// TIA Portal project "LAVADER0 DE COCHES" (V11)

(* hardware
DEVICE "S7300/ET200 station_1"  SIMATIC 300-Station
   slot 0: "Perfil soporte_0"  Rail  6ES7 390-1***0-0AA0
   slot 2: "PLC_1"  CPU 313C-2 DP  6ES7 313-6CF03-0AB0  V2.6
      slot 0: "Interfaz MPI_1"  MPI
      slot 1: "Interfaz DP_1"  DP
      slot 2: "DI16/DO16_1"  DI16/DO16
      slot 4: "Contaje_1"  Counter
DEVICE "S7300/ET200 station_2"  SIMATIC 300-Station
   slot 0: "Perfil soporte_0"  Rail  6ES7 390-1***0-0AA0
   slot 2: "JAVA"  CPU 313C-2 DP  6ES7 313-6CF03-0AB0  V2.6
      slot 0: "Interfaz MPI_1"  MPI
      slot 1: "Interfaz DP_1"  DP
      slot 2: "DI16/DO16_1"  DI16/DO16
      slot 4: "Contaje_1"  Counter
*)

// ===== PLC "PLC_1"  CPU 313C-2 DP =====

VAR_GLOBAL   // PLC tag table "Tabla de variables estándar"
   "M1 KM1 D ARRASTRE LENTA" AT %A0.0 : Bool;
   "M1 KM2 D ARRASTRE RAPIDA" AT %A0.1 : Bool;
   "M1 KM3 COMUN RAPIDA" AT %A0.2 : Bool;
   "M1 KM4 I RETROCESO LENTA" AT %A0.3 : Bool;
   "M1 KM5 I RETROCESO RAPIDA" AT %A0.4 : Bool;
   "M2 D VERTICAL" AT %A0.5 : Bool;
   "M2 I VERTICAL" AT %A0.6 : Bool;
   "M3 D HORIZONTAL" AT %A0.7 : Bool;
   "M3 I HORIZONTAL" AT %A1.0 : Bool;
   "M4 D LAVADO RUEDAS" AT %A1.1 : Bool;
   "M4 I LAVADO RUEDAS" AT %A1.2 : Bool;
   "VENTILADOR LINEA" AT %A1.3 : Bool;
   "VENTILADOE ESTRELLA" AT %A1.4 : Bool;
   "VENTILDOR TRIANGULO" AT %A1.5 : Bool;
   "BOMBA AGUA" AT %A1.6 : Bool;
   "BOMBA AIRE" AT %A1.7 : Bool;
   "BOMBA CHAMPU" AT %A2.0 : Bool;
   "tag_18" AT %E0.0 : Bool;
   "tag_19" AT %E0.1 : Bool;
   "tag_20" AT %E0.2 : Bool;
   "tag_21" AT %E0.3 : Bool;
   "Tag_22" AT %E0.4 : Bool;
   "Tag_23" AT %E0.5 : Bool;
   "Tag_24" AT %E0.6 : Bool;
   "Tag_25" AT %E0.7 : Bool;
   "Tag_26" AT %E1.0 : Bool;
   "Tag_27" AT %E1.1 : Bool;
   "Tag_28" AT %E1.2 : Bool;
   "Tag_29" AT %E1.3 : Bool;
   "Tag_30" AT %E1.4 : Bool;
   "Tag_31" AT %E1.5 : Bool;
   "Tag_32" AT %E1.6 : Bool;
   "Tag_33" AT %E1.7 : Bool;
   "tag_34" AT %E2.0 : Bool;
   "BOMBA CERA" AT %A2.1 : Bool;
   "PISTON VERTICAL" AT %A2.2 : Bool;
   "PISTON HORIZONTAL" AT %A2.3 : Bool;
   "PISTON L RUEDAS" AT %A2.4 : Bool;
   "Tag_39" AT %M0.0 : Bool;
   "Tag_1" AT %M0.3 : Bool;
   "Tag_2" AT %M0.4 : Bool;
   "Tag_3" AT %M0.5 : Bool;
   "Tag_4" AT %M0.6 : Bool;
   "Tag_5" AT %M0.7 : Bool;
   "Tag_6" AT %A11.5 : Bool;
   "Tag_7" AT %M8.0 : Bool;
   "Tag_8" AT %M10.0 : Bool;
   "Tag_9" AT %M10.1 : Bool;
   "Tag_10" AT %E2.2 : Bool;
   "V V EXPANDIDO" AT %A2.5 : Bool;
   "V V CONTRAIDO" AT %A2.6 : Bool;
   "V V SEMICONTRIDO" AT %A2.7 : Bool;
END_VAR

DATA_BLOCK "LAVADERO_DB"   // DB1
{ S7_Optimized_Access := 'FALSE' }
VERSION : 0.1
// stored: InstanceOfName LAVADERO
"LAVADERO"
BEGIN
   SWITCH[0] := 16#0;
   SW_SQTS[0] := 16#19;
   SW_SQTS[1] := 16#0;
   SW_SQTS[2] := 16#1;
   SW_SQTS[3] := 16#2;
   SW_SQTS[4] := 16#3;
   TVX[0] := 16#1;
   TTX[0] := 16#1;
   TSX[0] := 16#1;
   S00X[0] := 16#1;
   SOFFX[0] := 16#1;
   SONX[0] := 16#1;
   SAX[0] := 16#1;
   SERRX[0] := 16#1;
   SMX[0] := 16#1;
   S0X[0] := 16#1;
   S1X[0] := 16#1;
   SINI[0] := 16#2;
   SINI[1] := 16#1;
   LSTT[6] := 0;
   LSTT[5] := 16#1;
   ATAJ[1] := 16#1;
   ATAJ[2] := 16#2;
   ATAJ[3] := 16#3;
   ATAJ[4] := 16#4;
   ATAJ[5] := 16#5;
   ATAJ[6] := 16#6;
   ATAB[1] := 16#1B;
   ATAB[2] := 16#3;
   ATAB[3] := 16#1;
   ATAB[4] := 16#4;
   ATAB[5] := 16#5;
   ATAB[6] := 16#7;
   PSTT[1] := 16#1;
   PSTT[2] := 16#1;
   PSTT[3] := 16#1;
   PSTT[4] := 16#2;
   PSTT[5] := 16#3;
   PSTT[6] := 16#4;
   NSTT[0] := 16#1;
   NSTT[1] := 16#4;
   NSTT[2] := 16#2;
   NSTT[3] := 16#3;
   NSTT[4] := 16#1;
   NSTT[5] := 16#1;
   NSTT[6] := 16#5;
   ASSJ[1] := 16#1;
   ASSJ[2] := 16#2;
   ASSJ[3] := 16#3;
   ASSJ[4] := 16#4;
   ASSB[1] := 16#1;
   ASSB[2] := 16#2;
   ASSB[3] := 16#3;
   ASSB[4] := 16#4;
   PTTS[1] := 16#0;
   PTTS[2] := 16#2;
   PTTS[3] := 16#3;
   PTTS[4] := 16#1;
   NTTS[1] := 16#1;
   NTTS[2] := 16#4;
   NTTS[3] := 16#5;
   NTTS[4] := 16#6;
   LSTT[4] := 16#1;
   ATAJ[7] := 16#7;
   ATAB[7] := 16#6;
   PSTT[7] := 16#4;
   NSTT[7] := 16#1;
   SW_SQTS[5] := 16#4;
   ASSJ[5] := 16#5;
   ASSB[5] := 16#B;
   PTTS[5] := 16#6;
   NTTS[5] := 16#A;
   LSTT[7] := 16#1;
   SWITCH[1] := 16#0;
   SW_SQTS[6] := 16#5;
   SW_SQTS[7] := 16#6;
   LSTT[9] := 0;
   LSTT[10] := 0;
   ATAJ[8] := 16#8;
   ATAJ[9] := 16#9;
   ATAJ[10] := 16#A;
   ATAB[8] := 16#14;
   ATAB[9] := 16#D;
   ATAB[10] := 16#C;
   PSTT[8] := 16#8;
   PSTT[9] := 16#6;
   PSTT[10] := 16#5;
   NSTT[8] := 16#F;
   NSTT[9] := 16#7;
   NSTT[10] := 16#6;
   ASSJ[6] := 16#6;
   ASSJ[7] := 16#7;
   ASSB[6] := 16#6;
   ASSB[7] := 16#7;
   PTTS[6] := 16#A;
   PTTS[7] := 16#9;
   NTTS[6] := 16#9;
   NTTS[7] := 16#B;
   LSTT[11] := 0;
   ATAJ[11] := 16#B;
   ATAB[11] := 16#F;
   PSTT[11] := 16#7;
   NSTT[11] := 16#8;
   ATAJ[12] := 16#C;
   ATAB[12] := 16#A;
   PSTT[12] := 16#5;
   NSTT[12] := 16#1;
   LSTT[8] := 0;
   SW_SQTS[8] := 16#7;
   ASSJ[8] := 16#8;
   ASSB[8] := 16#8;
   PTTS[8] := 16#B;
   NTTS[8] := 16#8;
   LSTT[12] := 16#1;
   SWITCH[2] := 16#0;
   SW_SQTS[9] := 16#8;
   ATAJ[13] := 16#D;
   ATAB[13] := 16#9;
   PSTT[13] := 16#6;
   NSTT[13] := 16#1;
   ASSJ[9] := 16#9;
   ASSB[9] := 16#9;
   PTTS[9] := 16#E;
   NTTS[9] := 16#11;
   SWITCH[3] := 16#400106;
   SW_SQTS[10] := 16#9;
   LSTT[15] := 16#1;
   LSTT[16] := 16#1;
   LSTT[18] := 0;
   LSTT[19] := 16#13;
   ATAJ[14] := 16#E;
   ATAJ[15] := 16#F;
   ATAJ[16] := 16#10;
   ATAJ[17] := 16#11;
   ATAJ[18] := 16#12;
   ATAJ[19] := 16#13;
   ATAB[14] := 16#10;
   ATAB[15] := 16#B;
   ATAB[16] := 16#E;
   ATAB[17] := 16#15;
   ATAB[18] := 16#20;
   ATAB[19] := 16#17;
   PSTT[14] := 16#F;
   PSTT[15] := 16#7;
   PSTT[16] := 16#F;
   PSTT[17] := 16#9;
   PSTT[18] := 16#12;
   PSTT[19] := 16#C;
   NSTT[14] := 16#9;
   NSTT[15] := 16#1;
   NSTT[16] := 16#1;
   NSTT[17] := 16#A;
   NSTT[18] := 16#C;
   NSTT[19] := 16#13;
   ASSJ[10] := 16#A;
   ASSB[10] := 16#A;
   PTTS[10] := 16#11;
   NTTS[10] := 16#1F;
   SWITCH[4] := 16#80020C00;
   SW_SQTS[11] := 16#A;
   SW_SQTS[12] := 16#B;
   SW_SQTS[13] := 16#C;
   ATAJ[20] := 16#14;
   ATAJ[21] := 16#15;
   ATAB[20] := 16#8;
   ATAB[21] := 16#11;
   PSTT[20] := 16#8;
   PSTT[21] := 16#9;
   NSTT[20] := 16#1;
   NSTT[21] := 16#1;
   ASSJ[11] := 16#B;
   ASSJ[12] := 16#C;
   ASSJ[13] := 16#D;
   ASSB[11] := 16#16;
   ASSB[12] := 16#C;
   ASSB[13] := 16#D;
   PTTS[11] := 16#6;
   PTTS[12] := 16#12;
   PTTS[13] := 16#18;
   NTTS[11] := 16#18;
   NTTS[12] := 16#13;
   NTTS[13] := 16#19;
   SWITCH[5] := 16#518000A;
   SWITCH[6] := 16#30001460;
   SW_SQTS[14] := 16#D;
   LSTT[23] := 16#1;
   LSTT[24] := 0;
   LSTT[25] := 16#B;
   ATAJ[22] := 16#16;
   ATAJ[23] := 16#17;
   ATAJ[24] := 16#18;
   ATAJ[25] := 16#19;
   ATAB[22] := 16#1F;
   ATAB[23] := 16#13;
   ATAB[24] := 16#1A;
   ATAB[25] := 16#19;
   PSTT[22] := 16#A;
   PSTT[23] := 16#C;
   PSTT[24] := 16#B;
   PSTT[25] := 16#D;
   NSTT[22] := 16#1;
   NSTT[23] := 16#1;
   NSTT[24] := 16#D;
   NSTT[25] := 16#B;
   ASSJ[14] := 16#E;
   ASSB[14] := 16#10;
   PTTS[14] := 16#22;
   NTTS[14] := 16#1C;
   SWITCH[7] := 16#28C0C0;
   SW_SQTS[15] := 16#E;
   ATAJ[26] := 16#1A;
   ATAB[26] := 16#18;
   PSTT[26] := 16#B;
   NSTT[26] := 16#1;
   ASSJ[15] := 16#F;
   ASSB[15] := 16#F;
   PTTS[15] := 16#8;
   NTTS[15] := 16#E;
   LSTT[27] := 0;
   ATAJ[27] := 16#1B;
   ATAB[27] := 16#2;
   PSTT[27] := 16#1;
   NSTT[27] := 16#13;
   SW_SQTS[16] := 16#F;
   ATAJ[28] := 16#1C;
   ATAB[28] := 16#2C;
   PSTT[28] := 16#E;
   NSTT[28] := 16#14;
   ASSJ[16] := 16#10;
   ASSB[16] := 16#18;
   PTTS[16] := 16#22;
   NTTS[16] := 16#1D;
   LSTT[29] := 0;
   ATAJ[29] := 16#1D;
   ATAB[29] := 16#21;
   PSTT[29] := 16#10;
   NSTT[29] := 16#11;
   LSTT[26] := 16#1;
   LSTT[30] := 16#10;
   ATAJ[30] := 16#1E;
   ATAB[30] := 16#1E;
   PSTT[30] := 16#11;
   NSTT[30] := 16#10;
   SWITCH[8] := 16#2F8901A0;
   SWITCH[9] := 16#3BF24;
   SW_SQTS[17] := 16#10;
   LSTT[32] := 16#1;
   ATAJ[31] := 16#1F;
   ATAJ[32] := 16#20;
   ATAB[31] := 16#16;
   ATAB[32] := 16#12;
   PSTT[31] := 16#A;
   PSTT[32] := 16#12;
   NSTT[31] := 16#12;
   NSTT[32] := 16#1;
   ASSJ[17] := 16#11;
   ASSB[17] := 16#11;
   PTTS[17] := 16#1D;
   NTTS[17] := 16#1E;
   SW_SQTS[18] := 16#11;
   LSTT[17] := 0;
   LSTT[20] := 16#1;
   LSTT[28] := 0;
   LSTT[31] := 0;
   LSTT[33] := 16#1;
   ATAJ[33] := 16#21;
   ATAB[33] := 16#1D;
   PSTT[33] := 16#10;
   NSTT[33] := 16#1;
   ASSJ[18] := 16#12;
   ASSB[18] := 16#12;
   PTTS[18] := 16#1F;
   NTTS[18] := 16#12;
   SWITCH[10] := 16#6003030;
   LSTT[34] := 0;
   ATAJ[34] := 16#22;
   ATAB[34] := 16#23;
   PSTT[34] := 16#13;
   NSTT[34] := 16#E;
   SWITCH[11] := 16#51800;
   SW_SQTS[19] := 16#12;
   SW_SQTS[20] := 16#13;
   LSTT[36] := 16#1;
   LSTT[37] := 0;
   ATAJ[35] := 16#23;
   ATAJ[36] := 16#24;
   ATAJ[37] := 16#25;
   ATAB[35] := 16#22;
   ATAB[36] := 16#24;
   ATAB[37] := 16#2D;
   PSTT[35] := 16#13;
   PSTT[36] := 16#15;
   PSTT[37] := 16#14;
   NSTT[35] := 16#1;
   NSTT[36] := 16#1;
   NSTT[37] := 16#15;
   ASSJ[19] := 16#13;
   ASSJ[20] := 16#14;
   ASSB[19] := 16#13;
   ASSB[20] := 16#14;
   PTTS[19] := 16#1B;
   PTTS[20] := 16#1C;
   NTTS[19] := 16#22;
   NTTS[20] := 16#25;
   SW_SQTS[21] := 16#14;
   ATAJ[38] := 16#26;
   ATAB[38] := 16#28;
   PSTT[38] := 16#16;
   NSTT[38] := 16#17;
   ASSJ[21] := 16#15;
   ASSB[21] := 16#15;
   PTTS[21] := 16#25;
   NTTS[21] := 16#24;
   SWITCH[12] := 16#10CC0020;
   SWITCH[13] := 16#980128C0;
   LSTT[38] := 0;
   LSTT[39] := 16#16;
   ATAJ[39] := 16#27;
   ATAB[39] := 16#27;
   PSTT[39] := 16#17;
   NSTT[39] := 16#16;
   SW_SQTS[22] := 16#15;
   SW_SQTS[23] := 16#16;
   LSTT[40] := 16#1;
   ATAJ[40] := 16#28;
   ATAB[40] := 16#26;
   PSTT[40] := 16#16;
   NSTT[40] := 16#1;
   ASSJ[22] := 16#16;
   ASSJ[23] := 16#17;
   ASSB[22] := 16#5;
   ASSB[23] := 16#17;
   PTTS[22] := 16#6;
   PTTS[23] := 16#26;
   NTTS[22] := 16#26;
   NTTS[23] := 16#27;
   LSTT[35] := 16#1;
   LSTT[22] := 16#1;
   LSTT[21] := 16#1;
   LSTT[13] := 16#1;
   SWITCH[14] := 16#0;
   SWITCH[15] := 16#C0C00;
   SWITCH[16] := 16#1818FE4B;
   SW_SQTS[24] := 16#17;
   SW_SQTS[25] := 16#18;
   LSTT[42] := 16#18;
   LSTT[43] := 16#1;
   ATAJ[41] := 16#29;
   ATAJ[42] := 16#2A;
   ATAJ[43] := 16#2B;
   ATAB[41] := 16#2B;
   ATAB[42] := 16#2A;
   ATAB[43] := 16#29;
   PSTT[41] := 16#18;
   PSTT[42] := 16#19;
   PSTT[43] := 16#18;
   NSTT[41] := 16#19;
   NSTT[42] := 16#18;
   NSTT[43] := 16#1;
   ASSJ[24] := 16#18;
   ASSJ[25] := 16#19;
   ASSB[24] := 16#E;
   ASSB[25] := 16#19;
   PTTS[24] := 16#22;
   PTTS[25] := 16#29;
   NTTS[24] := 16#29;
   NTTS[25] := 16#2A;
   SWITCH[17] := 16#FC9700;
   SWITCH[18] := 16#D00C00;
   SWITCH[19] := 16#A0190000;
   LSTT[44] := 16#1;
   LSTT[45] := 16#1;
   ATAJ[44] := 16#2C;
   ATAJ[45] := 16#2D;
   ATAB[44] := 16#1C;
   ATAB[45] := 16#25;
   PSTT[44] := 16#E;
   PSTT[45] := 16#14;
   NSTT[44] := 16#1;
   NSTT[45] := 16#1;
END_DATA_BLOCK

FUNCTION_BLOCK "LAVADERO"   // FB1, GRAPH
{ S7_Optimized_Access := 'FALSE' }
VERSION : 0.1
   VAR_INPUT
      OFF_SQ : Bool := false;   // Desconectar cadena
      INIT_SQ : Bool := false;   // Poner cadena en estado inicial
      ACK_EF : Bool := false;   // Acusar todos los errores y fallos
      S_PREV : Bool := false;   // Mostrar la etapa anterior en el parámetro S_NO
      S_NEXT : Bool := false;   // Mostrar la etapa siguiente en el parámetro S_NO
      SW_AUTO : Bool := false;   // Modo automático
      SW_TAP : Bool := false;   // Semiautomático/continuar con transición
      SW_TOP : Bool := false;   // Semiautomático/transición ignorada
      SW_MAN : Bool := false;   // Modo manual
      S_SEL : Int := 0;   // Seleccionar la etapa que debe mostrarse en S_NO
      S_ON : Bool := false;   // Activar la etapa del parámetro S_NO
      S_OFF : Bool := false;   // Desactivar el incremento presente en el parámetro S_NO
      T_PUSH : Bool := false;   // Habilitar transición en modo semiautomático
      MICRO : Bool;
      SETA : Bool;
      EMERGENCIA : Bool;
      LLAVE : Bool;
      "A.CEPILLOS" : Bool;
      "S CEPILLOS" : Bool;
      "ABANCE CARRO" : Bool;
      "RETROCESO CARRO" : Bool;
      "FC LEVA" : Bool;
      "FC ABANCE" : Bool;
      "FC RETOCESO" : Bool;
      "FC VARILLA 1" : Bool;
      "SENSOR METALICO" : Bool;
      CLINOMETRO : Bool;
      CELULA : Bool;
   END_VAR
   VAR_OUTPUT
      S_NO : Int := 0;   // Número de etapa
      S_MORE : Bool := false;   // Existen más etapas que pueden mostrarse en S_NO.
      S_ACTIVE : Bool := false;   // El incremento presente en el parámetro S_NO está activo
      ERR_FLT : Bool := false;   // Error de grupo interlock o supervisión
      AUTO_ON : Bool := false;   // Modo automático activado
      TAP_ON : Bool := false;   // Modo semiautomático/etapa con transición activada
      TOP_ON : Bool := false;   // Modo semiautomático/Ignorar transición activado
      MAN_ON : Bool := false;   // Modo manual activado
      "M1 KM1 D ARRASTRE LENTA" : Bool;
      "M1 KM2 D ARRASTRE RAPIDA" : Bool;
      "M1 KM3 COMUN RAPIDA" : Bool;
      "M1 KM4 I RETROCESO LENTA" : Bool;
      "M1 KM5 I RETROCESO RAPIDA" : Bool;
      "M2 D VERTICAL" : Bool;
      "M2 I VERTICAL" : Bool;
      "M3 D HORIZONTAL" : Bool;
      "M3 I HORIZONTAL" : Bool;
      "M4 D LAVADO RUEDAS" : Bool;
      "M4 I LAVADO RUEDAS" : Bool;
      "VENTILADOR LINEA" : Bool;
      "VENTILADOR ESTRELLA" : Bool;
      "VENTILADOR TRIANULO" : Bool;
      "BOMBA AGUA" : Bool;
      "BOMBA AIRE" : Bool;
      "BOMBA CHAMPU" : Bool;
      "BOMBA CERA" : Bool;
      "PISTON VERTICAL" : Bool;
      "PISTON HORIZONAL" : Bool;
      "PISTON L RUEDAS" : Bool;
      "V V  EXPANDIDO" : Bool;
      "V V  CONTRAIDO" : Bool;
      "V V SEMICONTRAIDO" : Bool;
   END_VAR
   VAR
      SWITCH : Array [0..19]of DWord;
      SW_SQTS : Array [0..25]of Byte;
      SW_ADDR : Word := 16#E;
      G7T_0 : GraphTransition;
      G7S_0 : GraphStep;
      PRE_CRIT : Array [0..0]of DWord;
      POST_CRIT : Array [0..0]of DWord;
      TVX : Array [0..46]of Byte;
      TTX : Array [0..46]of Byte;
      TSX : Array [0..8]of Byte;
      S00X : Array [0..8]of Byte;
      SOFFX : Array [0..8]of Byte;
      SONX : Array [0..8]of Byte;
      SAX : Array [0..8]of Byte;
      SERRX : Array [0..26]of Byte;
      SMX : Array [0..26]of Byte;
      S0X : Array [0..26]of Byte;
      S1X : Array [0..26]of Byte;
      S_DISPLAY : Int;   // Indicación interna del parámetro de salida S_NO
      S_SEL_OLD : Int;   // Valor anterior en S_SEL
      S_DISPIDX : Byte;   // Índice de la etapa presente en S_NO
      T_DISPIDX : Byte;   // Índice de la transición presente en T_NO
      MOPEDGE : Struct
         AUTO : Bool := false;
         MAN : Bool := false;
         TAP : Bool := false;
         TOP : Bool := false;
         ACK_S : Bool := false;
         REG_S : Bool := false;
         T_PREV : Bool := false;
         T_NEXT : Bool := false;
         LOCK : Bool := false;
         SUP : Bool := false;
         ACKREQ : Bool := false;
         SSKIP : Bool := false;
         OFF : Bool := false;
         INIT : Bool := false;
         HALT : Bool := false;
         TMS_HALT : Bool := false;
         OPS_ZERO : Bool := false;
         SACT_DISP : Bool := false;
         SEF_DISP : Bool := false;
         SALL_DISP : Bool := false;
         S_PREV : Bool := false;
         S_NEXT : Bool := false;
         S_SELOK : Bool := false;
         S_ON : Bool := false;
         S_OFF : Bool := false;
         T_PUSH : Bool := false;
         REG : Bool := false;
         ACK : Bool := false;
         IL_PERM : Bool := false;
         T_PERM : Bool := false;
         ILP_MAN : Bool := false;
      END_STRUCT;
      MOP : Struct   // Modo de operación
         AUTO : Bool := true;   // Estado: modo automático
         MAN : Bool := false;   // Estado: modo manual
         TAP : Bool := false;   // Estado: semiautomático/continuar con transición
         TOP : Bool := false;   // Estado: semiautomático/transición ignorada
         ACK_S : Bool := false;   // Solicitud: acusar la etapa presente en el parámetro S_NO
         REG_S : Bool := false;   // Solicitud: registrar la etapa presente en el parámetro S_NO
         T_PREV : Bool := false;   // Solicitud: mostrar la transición anterior válida en el parámetro T_NO
         T_NEXT : Bool := false;   // Solicitud: mostrar la siguiente transición válida en el parámetro T_NO
         LOCK : Bool := true;   // Estado: ejecución de interlock activada
         SUP : Bool := true;   // Estado: ejecución de supervisión activada
         ACKREQ : Bool := true;   // Estado: acuse requerido
         SSKIP : Bool := false;   // Estado: "Saltar etapas" activado
         OFF : Bool := false;   // Solicitud: desactivar todas las etapas
         INIT : Bool := true;   // Solicitud: poner cadena en estado inicial
         HALT : Bool := false;   // Estado: la cadena no continúa
         TMS_HALT : Bool := false;   // Estado: todos los temporizadores internos detenidos
         OPS_ZERO : Bool := false;   // Estado: todos los operandos ejecutados con N, L, D puestos a 0
         SACT_DISP : Bool := true;   // Estado: mostrar sólo etapas activas
         SEF_DISP : Bool := false;   // Estado: mostrar sólo etapas erróneas y defectuosas
         SALL_DISP : Bool := false;   // Estado: mostrar todas las etapas
         S_PREV : Bool := false;   // Solicitud: mostrar la etapa anterior en el parámetro S_NO
         S_NEXT : Bool := false;   // Solicitud: Indicar etapa siguiente en el parámetro S_NO
         S_SELOK : Bool := false;   // Solicitud: mostrar en el parámetro S_NO el número de la etapa presente en el parámetro S_SEL
         S_ON : Bool := false;   // Solicitud: activar la etapa presente en el parámetro S_NO
         S_OFF : Bool := false;   // Solicitud: desactivar la etapa presente en el parámetro S_NO
         T_PUSH : Bool := false;   // Solicitud: habilitar transición
         REG : Bool := false;   // Solicitud: registrar todos los errores de interlock y supervisión
         ACK : Bool := false;   // Solicitud: acusar todos los errores de interlock y supervisión
         IL_PERM : Bool := false;   // Estado: ejecución permanente de todos los interlocks
         T_PERM : Bool := false;   // Estado: ejecución permanente de todas las transiciones
         ILP_MAN : Bool := false;   // Estado: ejecución permanente de todos los interlocks en modo manual
      END_STRUCT;
      TICKS : Struct   // Ciclos de tiempo
         DELTA : Time := T#0ms;   // Diferencia de tiempo entre dos ciclos
         OLD : Time := T#0ms;   // Estado de contador cíclico 10 ms en el último ciclo
         NEW : Time := T#0ms;   // Estado de contador cíclico 10 ms en este ciclo
      END_STRUCT;
      SQ_FLAGS : Struct   // Marcas de cadena
         ERR_FLT : Bool := false;   // Error de grupo interlock y supervisión
         ERROR : Bool := false;   // Error de grupo Interlock
         FAULT : Bool := false;   // Error de grupo Supervisión
         RT_FAIL : Bool := false;   // Error en tiempo de ejecución
         NO_SNO : Bool := false;   // No se ha encontrado el número de etapa solicitado
         NF_OFL : Bool := false;   // Desbordamiento: demasiadas solicitudes ON u OFF
         SA_OFL : Bool := false;   // Desbordamiento: demasiadas etapas activas
         TV_OFL : Bool := false;   // Desbordamiento: demasiadas transiciones válidas
         MSG_OFL : Bool := false;   // Desbordamiento: los recursos del sistema no son suficientes para ALARM_S
         NO_SWI : Bool := false;   // No conmutar en este ciclo
         CYC_OP : Bool := false;   // Ejecución cíclica de la cadena tras la inicialización
         AS_MSG : Bool := true;   // Avisos en tiempo de ejecución activados o desactivados por instrucción
         AS_SEND : Bool := false;   // Enviar avisos de WR_USMSG o sólo registrarlos en el búfer de diagnóstico
         SQ_BUSY : Bool := false;   // Marca de flanco interna para ejecución de proceso
         SA_BUSY : Bool := false;   // Marca de flanco interna para ejecución de proceso
         AS_SIG : Bool := false;   // Marca de flanco para avisos de Alarm_S y Alarm_SQ
      END_STRUCT;
      S_PTR : DWord := 16#1AD0;
      S_PTR2 : DWord := 16#0;
      S_PTR3 : DWord := 16#3C40;
      S_PTR4 : DWord := 16#3B60;
      T_PTR : DWord := 16#3A80;
      C_AR2 : DWord := 16#0;
      M_FBDB : DWord := 16#10000;
      M_SNO : Word := 16#0;
      M_EVID : Word := 16#0;
      M_EVIL : C_Alarm_s;
      M_EVSV : C_Alarm_s;
      M_EV : DWord := 16#38B0;
      CRIT : Array [0..31]of Bool;
      S_START : Byte := 16#0;
      S_IDX : Byte := 16#0;
      S_INT : Int := 72;
      S_TMP : Byte := 16#0;
      T_START : Byte := 16#0;
      T_IDX : Byte := 16#0;
      T_TMP : Byte := 16#0;
      T_TMP2 : Byte := 16#00;
      TV_POT : Byte := 16#08;
      RETURN1 : Byte := 16#0;
      RETURN2 : Byte := 16#0;
      SINI : Array [0..8]of Byte;
      LSTT : Array [0..45]of Byte;
      ATAJ : Array [0..45]of Byte;
      ATAB : Array [0..45]of Byte;
      PSTT : Array [0..45]of Byte;
      NSTT : Array [0..45]of Byte;
      ASSJ : Array [0..25]of Byte;
      ASSB : Array [0..25]of Byte;
      PTTS : Array [0..25]of Byte;
      NTTS : Array [0..25]of Byte;
      PRE_CNT : Word := 16#1;
      POST_CNT : Word := 16#1;
      ADR_COND : Word := 16#0;
      MAX_TVAL : Byte := 16#2D;
      MAX_SACT : Byte := 16#7;
      MAX_CRIT : Byte := 16#4;
      T_CNT : Byte := 16#2D;
      SUP_CNT : Byte := 16#0;
      LOCK_CNT : Byte := 16#6;
      S_CNT : Byte := 16#19;
      SQ_CNT : Byte := 16#1;
      PRS_INPAR : DWord := 16#E000FEC8;
      PRS_OUTPAR : DWord := 16#E000800F;
      GC_FLAGS : Struct
         T_MACH : Byte := 16#EB;
         COND_ED : Byte := 16#E3;
         W_LEVEL : Byte := 16#D5;
         FB_IF : Byte := 16#FA;
         AS_MSG : Word := 16#202;
         SSB : Word := 16#108;
         DILG : Word := 16#97C;
         ADDR_T0 : Word := 16#7A;
         CRIT_AVAIL : Bool := false;
         SSKIP_AVAIL : Bool := true;
         SSKIP_ON : Bool := false;
         ACK_REQ : Bool := true;
         SYNC_AVAIL : Bool := true;
         ILP_MAN : Bool := false;
         SWM_LOCKED : Bool := false;
         SAVE_SW : Bool := true;
      END_STRUCT;
      G7_FBMARK : Byte := 16#3C;
      G7_RELEASE : Byte := 16#3C;
      G7_ID2 : Byte := 16#37;
      G7_ID1 : Byte := 16#47;
   END_VAR
   // SWITCH[0] := 16#0;
   // SW_SQTS[0] := 16#19;
   // SW_SQTS[1] := 16#0;
   // SW_SQTS[2] := 16#1;
   // SW_SQTS[3] := 16#2;
   // SW_SQTS[4] := 16#3;
   // TVX[0] := 16#1;
   // TTX[0] := 16#1;
   // TSX[0] := 16#1;
   // S00X[0] := 16#1;
   // SOFFX[0] := 16#1;
   // SONX[0] := 16#1;
   // SAX[0] := 16#1;
   // SERRX[0] := 16#1;
   // SMX[0] := 16#1;
   // S0X[0] := 16#1;
   // S1X[0] := 16#1;
   // SINI[0] := 16#2;
   // SINI[1] := 16#1;
   // LSTT[6] := 0;
   // LSTT[5] := 16#1;
   // ATAJ[1] := 16#1;
   // ATAJ[2] := 16#2;
   // ATAJ[3] := 16#3;
   // ATAJ[4] := 16#4;
   // ATAJ[5] := 16#5;
   // ATAJ[6] := 16#6;
   // ATAB[1] := 16#1B;
   // ATAB[2] := 16#3;
   // ATAB[3] := 16#1;
   // ATAB[4] := 16#4;
   // ATAB[5] := 16#5;
   // ATAB[6] := 16#7;
   // PSTT[1] := 16#1;
   // PSTT[2] := 16#1;
   // PSTT[3] := 16#1;
   // PSTT[4] := 16#2;
   // PSTT[5] := 16#3;
   // PSTT[6] := 16#4;
   // NSTT[0] := 16#1;
   // NSTT[1] := 16#4;
   // NSTT[2] := 16#2;
   // NSTT[3] := 16#3;
   // NSTT[4] := 16#1;
   // NSTT[5] := 16#1;
   // NSTT[6] := 16#5;
   // ASSJ[1] := 16#1;
   // ASSJ[2] := 16#2;
   // ASSJ[3] := 16#3;
   // ASSJ[4] := 16#4;
   // ASSB[1] := 16#1;
   // ASSB[2] := 16#2;
   // ASSB[3] := 16#3;
   // ASSB[4] := 16#4;
   // PTTS[1] := 16#0;
   // PTTS[2] := 16#2;
   // PTTS[3] := 16#3;
   // PTTS[4] := 16#1;
   // NTTS[1] := 16#1;
   // NTTS[2] := 16#4;
   // NTTS[3] := 16#5;
   // NTTS[4] := 16#6;
   // LSTT[4] := 16#1;
   // ATAJ[7] := 16#7;
   // ATAB[7] := 16#6;
   // PSTT[7] := 16#4;
   // NSTT[7] := 16#1;
   // SW_SQTS[5] := 16#4;
   // ASSJ[5] := 16#5;
   // ASSB[5] := 16#B;
   // PTTS[5] := 16#6;
   // NTTS[5] := 16#A;
   // LSTT[7] := 16#1;
   // SWITCH[1] := 16#0;
   // SW_SQTS[6] := 16#5;
   // SW_SQTS[7] := 16#6;
   // LSTT[9] := 0;
   // LSTT[10] := 0;
   // ATAJ[8] := 16#8;
   // ATAJ[9] := 16#9;
   // ATAJ[10] := 16#A;
   // ATAB[8] := 16#14;
   // ATAB[9] := 16#D;
   // ATAB[10] := 16#C;
   // PSTT[8] := 16#8;
   // PSTT[9] := 16#6;
   // PSTT[10] := 16#5;
   // NSTT[8] := 16#F;
   // NSTT[9] := 16#7;
   // NSTT[10] := 16#6;
   // ASSJ[6] := 16#6;
   // ASSJ[7] := 16#7;
   // ASSB[6] := 16#6;
   // ASSB[7] := 16#7;
   // PTTS[6] := 16#A;
   // PTTS[7] := 16#9;
   // NTTS[6] := 16#9;
   // NTTS[7] := 16#B;
   // LSTT[11] := 0;
   // ATAJ[11] := 16#B;
   // ATAB[11] := 16#F;
   // PSTT[11] := 16#7;
   // NSTT[11] := 16#8;
   // ATAJ[12] := 16#C;
   // ATAB[12] := 16#A;
   // PSTT[12] := 16#5;
   // NSTT[12] := 16#1;
   // LSTT[8] := 0;
   // SW_SQTS[8] := 16#7;
   // ASSJ[8] := 16#8;
   // ASSB[8] := 16#8;
   // PTTS[8] := 16#B;
   // NTTS[8] := 16#8;
   // LSTT[12] := 16#1;
   // SWITCH[2] := 16#0;
   // SW_SQTS[9] := 16#8;
   // ATAJ[13] := 16#D;
   // ATAB[13] := 16#9;
   // PSTT[13] := 16#6;
   // NSTT[13] := 16#1;
   // ASSJ[9] := 16#9;
   // ASSB[9] := 16#9;
   // PTTS[9] := 16#E;
   // NTTS[9] := 16#11;
   // SWITCH[3] := 16#400106;
   // SW_SQTS[10] := 16#9;
   // LSTT[15] := 16#1;
   // LSTT[16] := 16#1;
   // LSTT[18] := 0;
   // LSTT[19] := 16#13;
   // ATAJ[14] := 16#E;
   // ATAJ[15] := 16#F;
   // ATAJ[16] := 16#10;
   // ATAJ[17] := 16#11;
   // ATAJ[18] := 16#12;
   // ATAJ[19] := 16#13;
   // ATAB[14] := 16#10;
   // ATAB[15] := 16#B;
   // ATAB[16] := 16#E;
   // ATAB[17] := 16#15;
   // ATAB[18] := 16#20;
   // ATAB[19] := 16#17;
   // PSTT[14] := 16#F;
   // PSTT[15] := 16#7;
   // PSTT[16] := 16#F;
   // PSTT[17] := 16#9;
   // PSTT[18] := 16#12;
   // PSTT[19] := 16#C;
   // NSTT[14] := 16#9;
   // NSTT[15] := 16#1;
   // NSTT[16] := 16#1;
   // NSTT[17] := 16#A;
   // NSTT[18] := 16#C;
   // NSTT[19] := 16#13;
   // ASSJ[10] := 16#A;
   // ASSB[10] := 16#A;
   // PTTS[10] := 16#11;
   // NTTS[10] := 16#1F;
   // SWITCH[4] := 16#80020C00;
   // SW_SQTS[11] := 16#A;
   // SW_SQTS[12] := 16#B;
   // SW_SQTS[13] := 16#C;
   // ATAJ[20] := 16#14;
   // ATAJ[21] := 16#15;
   // ATAB[20] := 16#8;
   // ATAB[21] := 16#11;
   // PSTT[20] := 16#8;
   // PSTT[21] := 16#9;
   // NSTT[20] := 16#1;
   // NSTT[21] := 16#1;
   // ASSJ[11] := 16#B;
   // ASSJ[12] := 16#C;
   // ASSJ[13] := 16#D;
   // ASSB[11] := 16#16;
   // ASSB[12] := 16#C;
   // ASSB[13] := 16#D;
   // PTTS[11] := 16#6;
   // PTTS[12] := 16#12;
   // PTTS[13] := 16#18;
   // NTTS[11] := 16#18;
   // NTTS[12] := 16#13;
   // NTTS[13] := 16#19;
   // SWITCH[5] := 16#518000A;
   // SWITCH[6] := 16#30001460;
   // SW_SQTS[14] := 16#D;
   // LSTT[23] := 16#1;
   // LSTT[24] := 0;
   // LSTT[25] := 16#B;
   // ATAJ[22] := 16#16;
   // ATAJ[23] := 16#17;
   // ATAJ[24] := 16#18;
   // ATAJ[25] := 16#19;
   // ATAB[22] := 16#1F;
   // ATAB[23] := 16#13;
   // ATAB[24] := 16#1A;
   // ATAB[25] := 16#19;
   // PSTT[22] := 16#A;
   // PSTT[23] := 16#C;
   // PSTT[24] := 16#B;
   // PSTT[25] := 16#D;
   // NSTT[22] := 16#1;
   // NSTT[23] := 16#1;
   // NSTT[24] := 16#D;
   // NSTT[25] := 16#B;
   // ASSJ[14] := 16#E;
   // ASSB[14] := 16#10;
   // PTTS[14] := 16#22;
   // NTTS[14] := 16#1C;
   // SWITCH[7] := 16#28C0C0;
   // SW_SQTS[15] := 16#E;
   // ATAJ[26] := 16#1A;
   // ATAB[26] := 16#18;
   // PSTT[26] := 16#B;
   // NSTT[26] := 16#1;
   // ASSJ[15] := 16#F;
   // ASSB[15] := 16#F;
   // PTTS[15] := 16#8;
   // NTTS[15] := 16#E;
   // LSTT[27] := 0;
   // ATAJ[27] := 16#1B;
   // ATAB[27] := 16#2;
   // PSTT[27] := 16#1;
   // NSTT[27] := 16#13;
   // SW_SQTS[16] := 16#F;
   // ATAJ[28] := 16#1C;
   // ATAB[28] := 16#2C;
   // PSTT[28] := 16#E;
   // NSTT[28] := 16#14;
   // ASSJ[16] := 16#10;
   // ASSB[16] := 16#18;
   // PTTS[16] := 16#22;
   // NTTS[16] := 16#1D;
   // LSTT[29] := 0;
   // ATAJ[29] := 16#1D;
   // ATAB[29] := 16#21;
   // PSTT[29] := 16#10;
   // NSTT[29] := 16#11;
   // LSTT[26] := 16#1;
   // LSTT[30] := 16#10;
   // ATAJ[30] := 16#1E;
   // ATAB[30] := 16#1E;
   // PSTT[30] := 16#11;
   // NSTT[30] := 16#10;
   // SWITCH[8] := 16#2F8901A0;
   // SWITCH[9] := 16#3BF24;
   // SW_SQTS[17] := 16#10;
   // LSTT[32] := 16#1;
   // ATAJ[31] := 16#1F;
   // ATAJ[32] := 16#20;
   // ATAB[31] := 16#16;
   // ATAB[32] := 16#12;
   // PSTT[31] := 16#A;
   // PSTT[32] := 16#12;
   // NSTT[31] := 16#12;
   // NSTT[32] := 16#1;
   // ASSJ[17] := 16#11;
   // ASSB[17] := 16#11;
   // PTTS[17] := 16#1D;
   // NTTS[17] := 16#1E;
   // SW_SQTS[18] := 16#11;
   // LSTT[17] := 0;
   // LSTT[20] := 16#1;
   // LSTT[28] := 0;
   // LSTT[31] := 0;
   // LSTT[33] := 16#1;
   // ATAJ[33] := 16#21;
   // ATAB[33] := 16#1D;
   // PSTT[33] := 16#10;
   // NSTT[33] := 16#1;
   // ASSJ[18] := 16#12;
   // ASSB[18] := 16#12;
   // PTTS[18] := 16#1F;
   // NTTS[18] := 16#12;
   // SWITCH[10] := 16#6003030;
   // LSTT[34] := 0;
   // ATAJ[34] := 16#22;
   // ATAB[34] := 16#23;
   // PSTT[34] := 16#13;
   // NSTT[34] := 16#E;
   // SWITCH[11] := 16#51800;
   // SW_SQTS[19] := 16#12;
   // SW_SQTS[20] := 16#13;
   // LSTT[36] := 16#1;
   // LSTT[37] := 0;
   // ATAJ[35] := 16#23;
   // ATAJ[36] := 16#24;
   // ATAJ[37] := 16#25;
   // ATAB[35] := 16#22;
   // ATAB[36] := 16#24;
   // ATAB[37] := 16#2D;
   // PSTT[35] := 16#13;
   // PSTT[36] := 16#15;
   // PSTT[37] := 16#14;
   // NSTT[35] := 16#1;
   // NSTT[36] := 16#1;
   // NSTT[37] := 16#15;
   // ASSJ[19] := 16#13;
   // ASSJ[20] := 16#14;
   // ASSB[19] := 16#13;
   // ASSB[20] := 16#14;
   // PTTS[19] := 16#1B;
   // PTTS[20] := 16#1C;
   // NTTS[19] := 16#22;
   // NTTS[20] := 16#25;
   // SW_SQTS[21] := 16#14;
   // ATAJ[38] := 16#26;
   // ATAB[38] := 16#28;
   // PSTT[38] := 16#16;
   // NSTT[38] := 16#17;
   // ASSJ[21] := 16#15;
   // ASSB[21] := 16#15;
   // PTTS[21] := 16#25;
   // NTTS[21] := 16#24;
   // SWITCH[12] := 16#10CC0020;
   // SWITCH[13] := 16#980128C0;
   // LSTT[38] := 0;
   // LSTT[39] := 16#16;
   // ATAJ[39] := 16#27;
   // ATAB[39] := 16#27;
   // PSTT[39] := 16#17;
   // NSTT[39] := 16#16;
   // SW_SQTS[22] := 16#15;
   // SW_SQTS[23] := 16#16;
   // LSTT[40] := 16#1;
   // ATAJ[40] := 16#28;
   // ATAB[40] := 16#26;
   // PSTT[40] := 16#16;
   // NSTT[40] := 16#1;
   // ASSJ[22] := 16#16;
   // ASSJ[23] := 16#17;
   // ASSB[22] := 16#5;
   // ASSB[23] := 16#17;
   // PTTS[22] := 16#6;
   // PTTS[23] := 16#26;
   // NTTS[22] := 16#26;
   // NTTS[23] := 16#27;
   // LSTT[35] := 16#1;
   // LSTT[22] := 16#1;
   // LSTT[21] := 16#1;
   // LSTT[13] := 16#1;
   // SWITCH[14] := 16#0;
   // SWITCH[15] := 16#C0C00;
   // SWITCH[16] := 16#1818FE4B;
   // SW_SQTS[24] := 16#17;
   // SW_SQTS[25] := 16#18;
   // LSTT[42] := 16#18;
   // LSTT[43] := 16#1;
   // ATAJ[41] := 16#29;
   // ATAJ[42] := 16#2A;
   // ATAJ[43] := 16#2B;
   // ATAB[41] := 16#2B;
   // ATAB[42] := 16#2A;
   // ATAB[43] := 16#29;
   // PSTT[41] := 16#18;
   // PSTT[42] := 16#19;
   // PSTT[43] := 16#18;
   // NSTT[41] := 16#19;
   // NSTT[42] := 16#18;
   // NSTT[43] := 16#1;
   // ASSJ[24] := 16#18;
   // ASSJ[25] := 16#19;
   // ASSB[24] := 16#E;
   // ASSB[25] := 16#19;
   // PTTS[24] := 16#22;
   // PTTS[25] := 16#29;
   // NTTS[24] := 16#29;
   // NTTS[25] := 16#2A;
   // SWITCH[17] := 16#FC9700;
   // SWITCH[18] := 16#D00C00;
   // SWITCH[19] := 16#A0190000;
   // LSTT[44] := 16#1;
   // LSTT[45] := 16#1;
   // ATAJ[44] := 16#2C;
   // ATAJ[45] := 16#2D;
   // ATAB[44] := 16#1C;
   // ATAB[45] := 16#25;
   // PSTT[44] := 16#E;
   // PSTT[45] := 16#14;
   // NSTT[44] := 16#1;
   // NSTT[45] := 16#1;
BEGIN
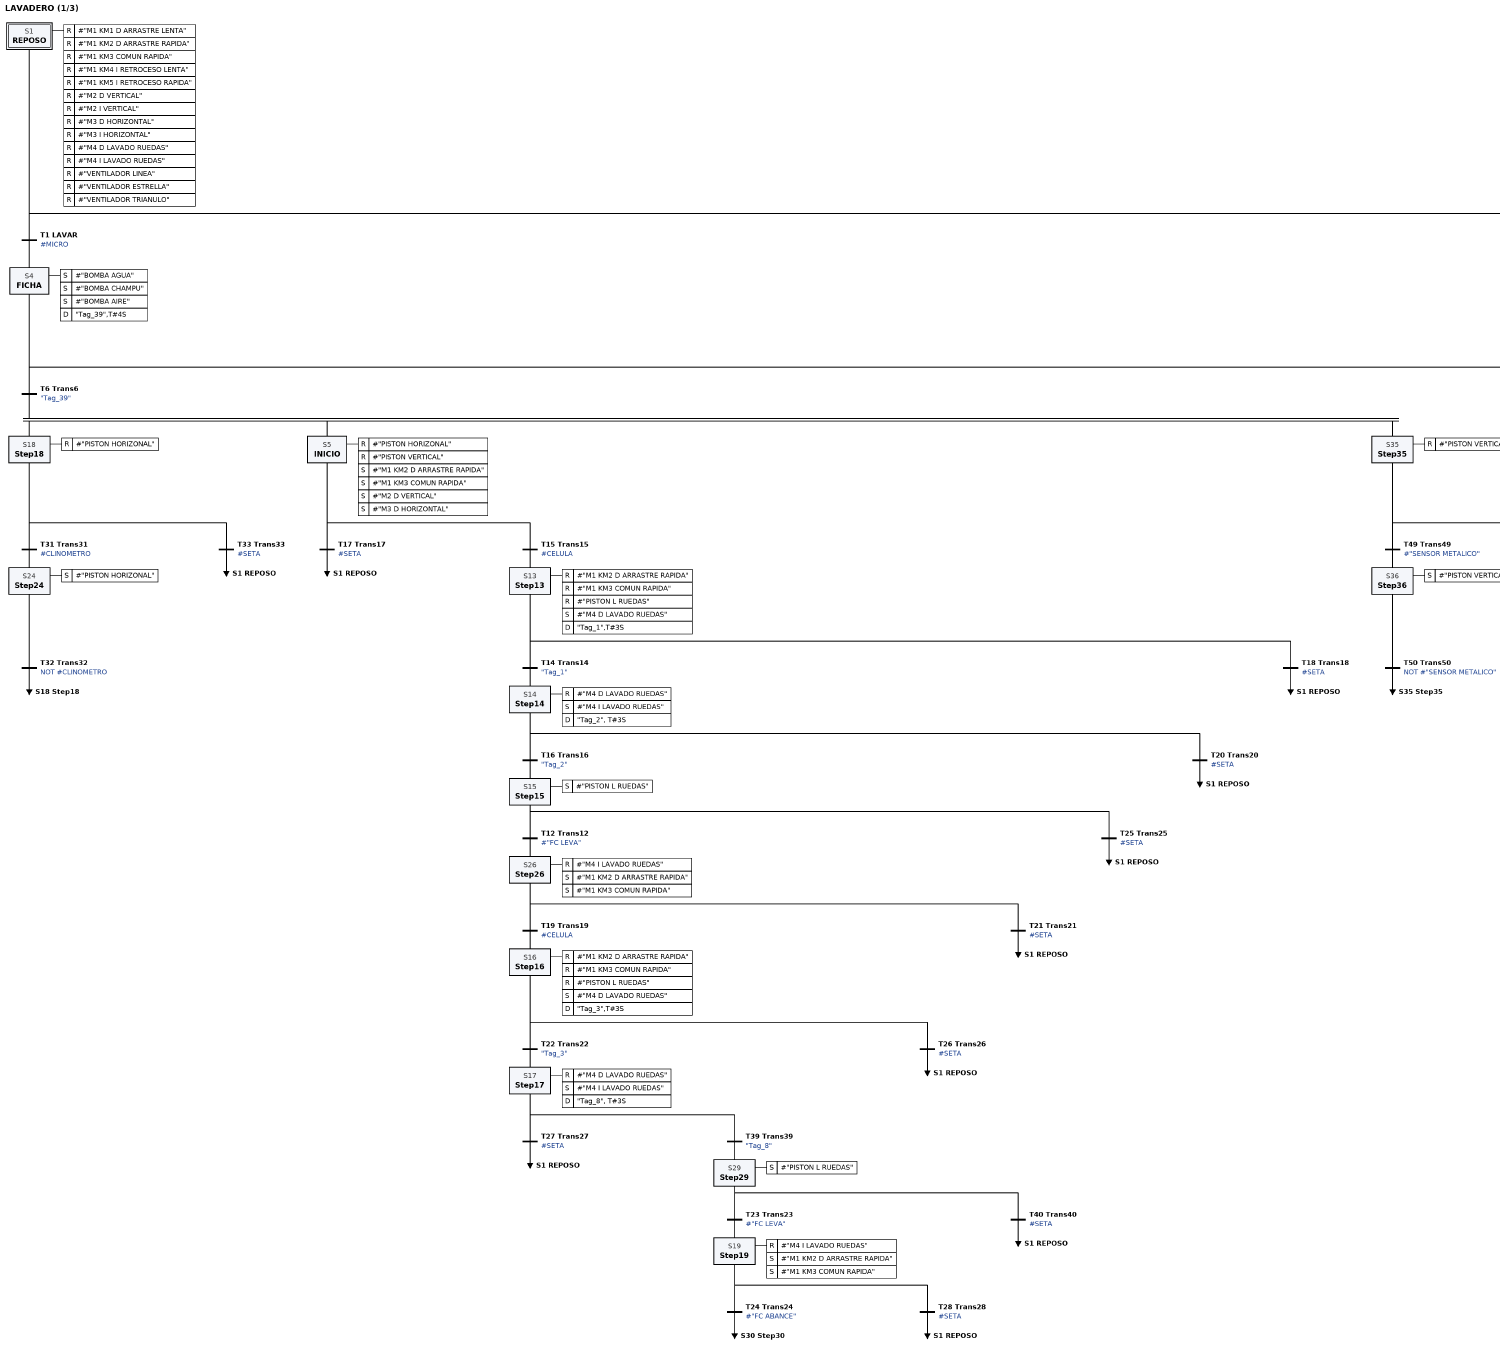
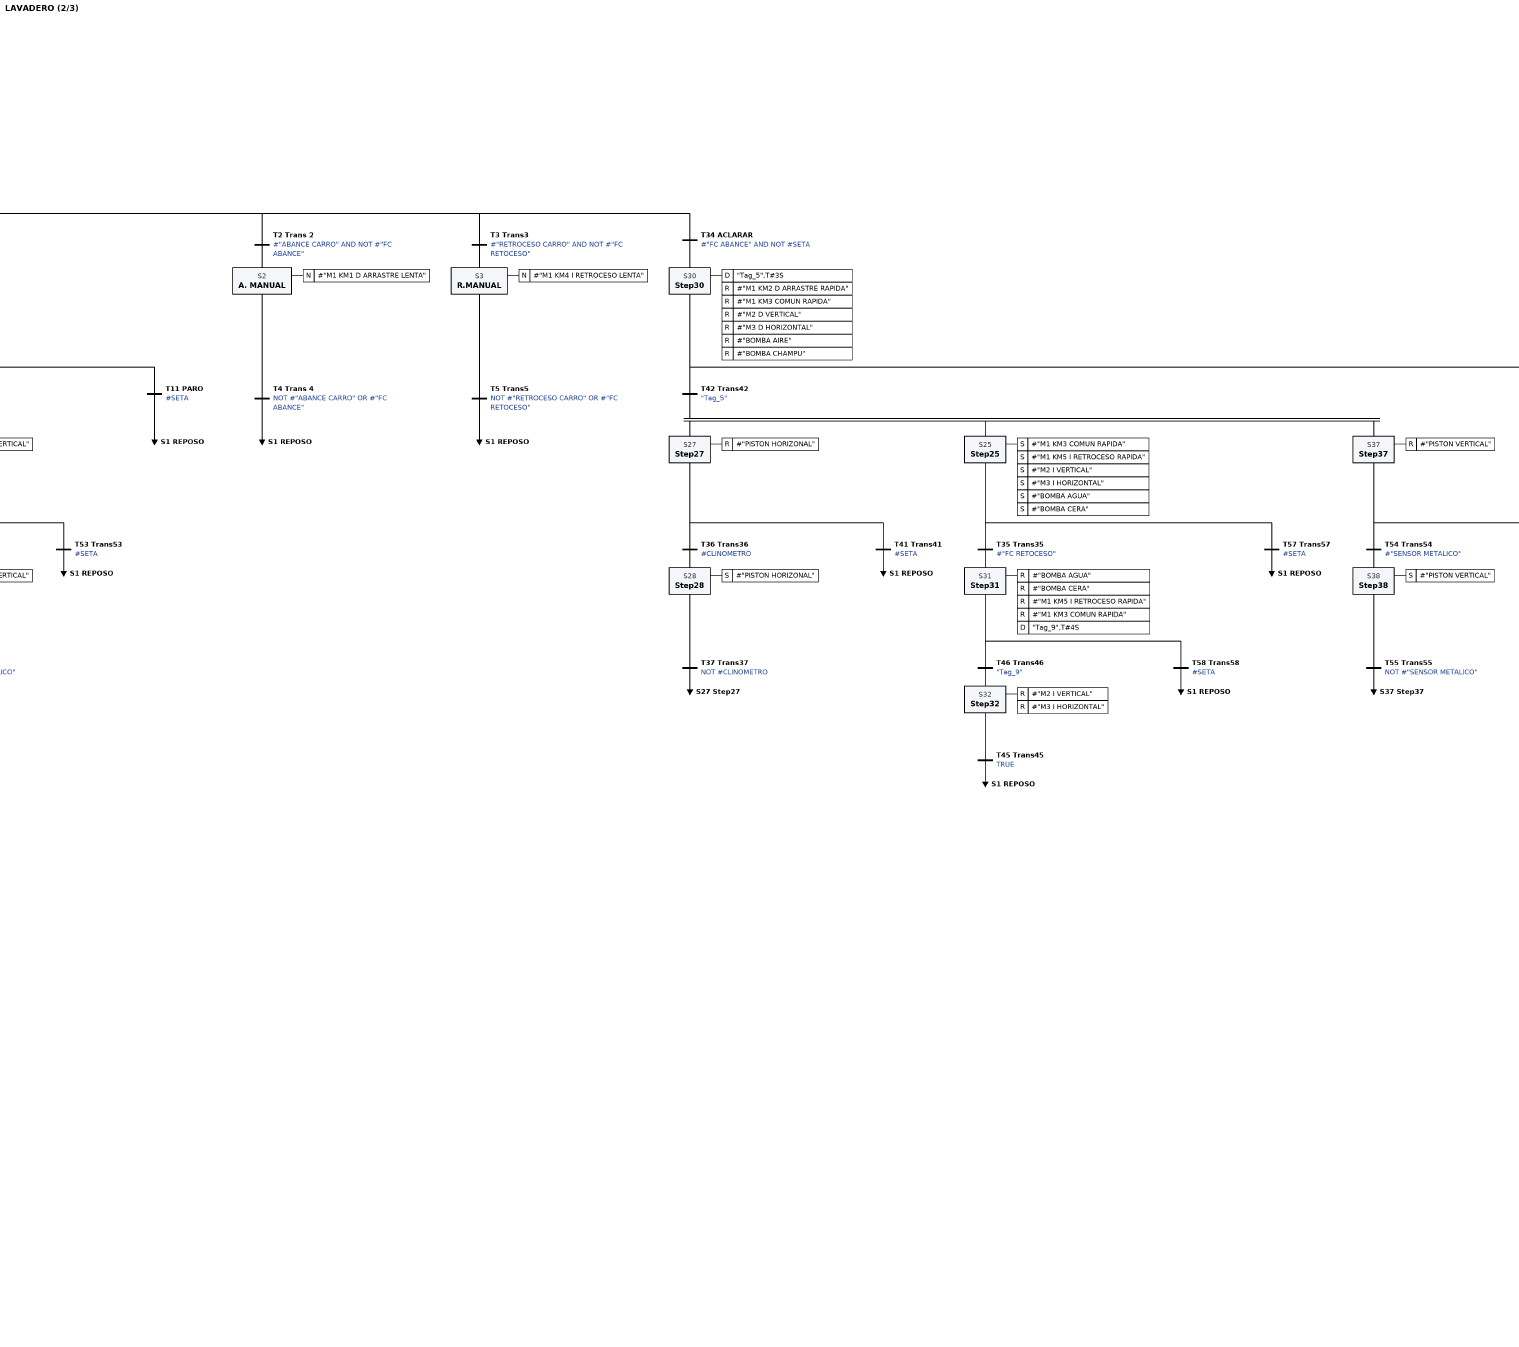
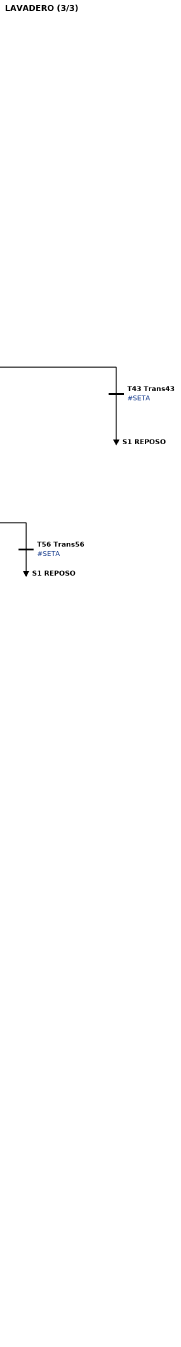
   // sequencer 1
   INITIAL_STEP REPOSO:   // S1
      // REPOSO .
              R    #"M1 KM1 D ARRASTRE LENTA"
              R    #"M1 KM2 D ARRASTRE RAPIDA"
              R    #"M1 KM3 COMUN RAPIDA"
              R    #"M1 KM4 I RETROCESO LENTA"
              R    #"M1 KM5 I RETROCESO RAPIDA"
              R    #"M2 D VERTICAL"
              R    #"M2 I VERTICAL"
              R    #"M3 D HORIZONTAL"
              R    #"M3 I HORIZONTAL"
              R    #"M4 D LAVADO RUEDAS"
              R    #"M4 I LAVADO RUEDAS"
              R    #"VENTILADOR LINEA"
              R    #"VENTILADOR ESTRELLA"
              R    #"VENTILADOR TRIANULO"
              R    #"BOMBA AGUA"
              R    #"BOMBA AIRE"
              R    #"BOMBA CHAMPU"
              R    #"BOMBA CERA"
              R    #"V V  CONTRAIDO"
              R    #"V V SEMICONTRAIDO"
              S    #"PISTON VERTICAL"
              S    #"PISTON HORIZONAL"
              S    #"PISTON L RUEDAS"
              S    #"V V  EXPANDIDO"
   END_STEP
   TRANSITION LAVAR FROM REPOSO TO FICHA   // T1: INTRODUCCION FICHA.
      := #MICRO;
   END_TRANSITION
   TRANSITION "Trans 2" FROM REPOSO TO "A. MANUAL"   // T2: ABANCE CARRO MANUAL POR PULSOS.
      := #"ABANCE CARRO" AND NOT #"FC ABANCE";
   END_TRANSITION
   TRANSITION Trans3 FROM REPOSO TO "R.MANUAL"   // T3: RETROCESO CARRO MANUAL POR PULSOS.
      := #"RETROCESO CARRO" AND NOT #"FC RETOCESO";
   END_TRANSITION
   TRANSITION ACLARAR FROM REPOSO TO Step30   // T34
      := #"FC ABANCE" AND NOT #SETA;
   END_TRANSITION
   STEP "A. MANUAL":   // S2
      interlock C := #"RETROCESO CARRO";
              N    #"M1 KM1 D ARRASTRE LENTA"
   END_STEP
   TRANSITION "Trans 4" FROM "A. MANUAL" TO REPOSO   // T4, jump
      := NOT #"ABANCE CARRO" OR #"FC ABANCE";
   END_TRANSITION
   STEP FICHA:   // S4
              S    #"BOMBA AGUA"
              S    #"BOMBA CHAMPU"
              S    #"BOMBA AIRE"
              D    "Tag_39",T#4S
   END_STEP
   TRANSITION Trans6 FROM FICHA TO (Step18, INICIO, Step35)   // T6
      := "Tag_39";
   END_TRANSITION
   TRANSITION PARO FROM FICHA TO REPOSO   // T11, jump
      := #SETA;
   END_TRANSITION
   STEP "R.MANUAL":   // S3
      interlock C := #"ABANCE CARRO";
              N    #"M1 KM4 I RETROCESO LENTA"
   END_STEP
   TRANSITION Trans5 FROM "R.MANUAL" TO REPOSO   // T5, jump
      := NOT #"RETROCESO CARRO" OR #"FC RETOCESO";
   END_TRANSITION
   STEP INICIO:   // S5
              R    #"PISTON HORIZONAL"
              R    #"PISTON VERTICAL"
              S    #"M1 KM2 D ARRASTRE RAPIDA"
              S    #"M1 KM3 COMUN RAPIDA"
              S    #"M2 D VERTICAL"
              S    #"M3 D HORIZONTAL"
   END_STEP
   TRANSITION Trans17 FROM INICIO TO REPOSO   // T17, jump
      := #SETA;
   END_TRANSITION
   TRANSITION Trans15 FROM INICIO TO Step13   // T15
      := #CELULA;
   END_TRANSITION
   STEP Step13:   // S13
              R    #"M1 KM2 D ARRASTRE RAPIDA"
              R    #"M1 KM3 COMUN RAPIDA"
              R    #"PISTON L RUEDAS"
              S    #"M4 D LAVADO RUEDAS"
              D    "Tag_1",T#3S
   END_STEP
   TRANSITION Trans14 FROM Step13 TO Step14   // T14
      := "Tag_1";
   END_TRANSITION
   TRANSITION Trans18 FROM Step13 TO REPOSO   // T18, jump
      := #SETA;
   END_TRANSITION
   STEP Step15:   // S15
              S    #"PISTON L RUEDAS"
   END_STEP
   TRANSITION Trans12 FROM Step15 TO Step26   // T12
      := #"FC LEVA";
   END_TRANSITION
   TRANSITION Trans25 FROM Step15 TO REPOSO   // T25, jump
      := #SETA;
   END_TRANSITION
   STEP Step14:   // S14
              R    #"M4 D LAVADO RUEDAS"
              S    #"M4 I LAVADO RUEDAS"
              D    "Tag_2", T#3S
   END_STEP
   TRANSITION Trans16 FROM Step14 TO Step15   // T16
      := "Tag_2";
   END_TRANSITION
   TRANSITION Trans20 FROM Step14 TO REPOSO   // T20, jump
      := #SETA;
   END_TRANSITION
   STEP Step16:   // S16
              R    #"M1 KM2 D ARRASTRE RAPIDA"
              R    #"M1 KM3 COMUN RAPIDA"
              R    #"PISTON L RUEDAS"
              S    #"M4 D LAVADO RUEDAS"
              D    "Tag_3",T#3S
   END_STEP
   TRANSITION Trans22 FROM Step16 TO Step17   // T22
      := "Tag_3";
   END_TRANSITION
   TRANSITION Trans26 FROM Step16 TO REPOSO   // T26, jump
      := #SETA;
   END_TRANSITION
   STEP Step17:   // S17
              R    #"M4 D LAVADO RUEDAS"
              S    #"M4 I LAVADO RUEDAS"
              D    "Tag_8", T#3S
   END_STEP
   TRANSITION Trans27 FROM Step17 TO REPOSO   // T27, jump
      := #SETA;
   END_TRANSITION
   TRANSITION Trans39 FROM Step17 TO Step29   // T39
      := "Tag_8";
   END_TRANSITION
   STEP Step18:   // S18
      interlock C := #CLINOMETRO;
              R    #"PISTON HORIZONAL"
   END_STEP
   TRANSITION Trans31 FROM Step18 TO Step24   // T31
      := #CLINOMETRO;
   END_TRANSITION
   TRANSITION Trans33 FROM Step18 TO REPOSO   // T33, jump
      := #SETA;
   END_TRANSITION
   STEP Step19:   // S19
              R    #"M4 I LAVADO RUEDAS"
              S    #"M1 KM2 D ARRASTRE RAPIDA"
              S    #"M1 KM3 COMUN RAPIDA"
   END_STEP
   TRANSITION Trans24 FROM Step19 TO Step30   // T24, jump
      := #"FC ABANCE";
   END_TRANSITION
   TRANSITION Trans28 FROM Step19 TO REPOSO   // T28, jump
      := #SETA;
   END_TRANSITION
   STEP Step30:   // S30
              D    "Tag_5",T#3S
              R    #"M1 KM2 D ARRASTRE RAPIDA"
              R    #"M1 KM3 COMUN RAPIDA"
              R    #"M2 D VERTICAL"
              R    #"M3 D HORIZONTAL"
              R    #"BOMBA AIRE"
              R    #"BOMBA CHAMPU"
   END_STEP
   TRANSITION Trans42 FROM Step30 TO (Step27, Step25, Step37)   // T42
      := "Tag_5";
   END_TRANSITION
   TRANSITION Trans43 FROM Step30 TO REPOSO   // T43, jump
      := #SETA;
   END_TRANSITION
   STEP Step24:   // S24
              S    #"PISTON HORIZONAL"
   END_STEP
   TRANSITION Trans32 FROM Step24 TO Step18   // T32, jump
      := NOT #CLINOMETRO;
   END_TRANSITION
   STEP Step25:   // S25
              S    #"M1 KM3 COMUN RAPIDA"
              S    #"M1 KM5 I RETROCESO RAPIDA"
              S    #"M2 I VERTICAL"
              S    #"M3 I HORIZONTAL"
              S    #"BOMBA AGUA"
              S    #"BOMBA CERA"
   END_STEP
   TRANSITION Trans35 FROM Step25 TO Step31   // T35
      := #"FC RETOCESO";
   END_TRANSITION
   TRANSITION Trans57 FROM Step25 TO REPOSO   // T57, jump
      := #SETA;
   END_TRANSITION
   STEP Step26:   // S26
              R    #"M4 I LAVADO RUEDAS"
              S    #"M1 KM2 D ARRASTRE RAPIDA"
              S    #"M1 KM3 COMUN RAPIDA"
   END_STEP
   TRANSITION Trans19 FROM Step26 TO Step16   // T19
      := #CELULA;
   END_TRANSITION
   TRANSITION Trans21 FROM Step26 TO REPOSO   // T21, jump
      := #SETA;
   END_TRANSITION
   STEP Step27:   // S27
      interlock C := #CLINOMETRO;
              R    #"PISTON HORIZONAL"
   END_STEP
   TRANSITION Trans36 FROM Step27 TO Step28   // T36
      := #CLINOMETRO;
   END_TRANSITION
   TRANSITION Trans41 FROM Step27 TO REPOSO   // T41, jump
      := #SETA;
   END_TRANSITION
   STEP Step28:   // S28
              S    #"PISTON HORIZONAL"
   END_STEP
   TRANSITION Trans37 FROM Step28 TO Step27   // T37, jump
      := NOT #CLINOMETRO;
   END_TRANSITION
   STEP Step29:   // S29
              S    #"PISTON L RUEDAS"
   END_STEP
   TRANSITION Trans23 FROM Step29 TO Step19   // T23
      := #"FC LEVA";
   END_TRANSITION
   TRANSITION Trans40 FROM Step29 TO REPOSO   // T40, jump
      := #SETA;
   END_TRANSITION
   STEP Step31:   // S31
              R    #"BOMBA AGUA"
              R    #"BOMBA CERA"
              R    #"M1 KM5 I RETROCESO RAPIDA"
              R    #"M1 KM3 COMUN RAPIDA"
              D    "Tag_9",T#4S
   END_STEP
   TRANSITION Trans46 FROM Step31 TO Step32   // T46
      := "Tag_9";
   END_TRANSITION
   TRANSITION Trans58 FROM Step31 TO REPOSO   // T58, jump
      := #SETA;
   END_TRANSITION
   STEP Step32:   // S32
              R    #"M2 I VERTICAL"
              R    #"M3 I HORIZONTAL"
   END_STEP
   TRANSITION Trans45 FROM Step32 TO REPOSO   // T45, jump
      := TRUE;
   END_TRANSITION
   STEP Step37:   // S37
      interlock C := #"SENSOR METALICO";
              R    #"PISTON VERTICAL"
   END_STEP
   TRANSITION Trans54 FROM Step37 TO Step38   // T54
      := #"SENSOR METALICO";
   END_TRANSITION
   TRANSITION Trans56 FROM Step37 TO REPOSO   // T56, jump
      := #SETA;
   END_TRANSITION
   STEP Step38:   // S38
              S    #"PISTON VERTICAL"
   END_STEP
   TRANSITION Trans55 FROM Step38 TO Step37   // T55, jump
      := NOT #"SENSOR METALICO";
   END_TRANSITION
   STEP Step35:   // S35
      interlock C := #"SENSOR METALICO";
              R    #"PISTON VERTICAL"
   END_STEP
   TRANSITION Trans49 FROM Step35 TO Step36   // T49
      := #"SENSOR METALICO";
   END_TRANSITION
   TRANSITION Trans53 FROM Step35 TO REPOSO   // T53, jump
      := #SETA;
   END_TRANSITION
   STEP Step36:   // S36
              S    #"PISTON VERTICAL"
   END_STEP
   TRANSITION Trans50 FROM Step36 TO Step35   // T50, jump
      := NOT #"SENSOR METALICO";
   END_TRANSITION
END_FUNCTION_BLOCK

ORGANIZATION_BLOCK "Main"   // OB1, LAD
TITLE = "Main Program Sweep (Cycle)"
{ S7_Optimized_Access := 'FALSE' }
VERSION : 0.1
   VAR_TEMP
      OB1_EV_CLASS : Byte;   // Bits 0-3 = 1 (Coming event), Bits 4-7 = 1 (Event class 1)
      OB1_SCAN_1 : Byte;   // 1 (Cold restart scan 1 of OB 1), 3 (Scan 2-n of OB 1)
      OB1_PRIORITY : Byte;   // Priority of OB Execution
      OB1_OB_NUMBR : Byte;   // 1 (Organization block 1, OB1)
      OB1_RESERVED_1 : Byte;   // Reserved for system
      OB1_RESERVED_2 : Byte;   // Reserved for system
      OB1_PREV_CYCLE : Int;   // Cycle time of previous OB1 scan (milliseconds)
      OB1_MIN_CYCLE : Int;   // Minimum cycle time of OB1 (milliseconds)
      OB1_MAX_CYCLE : Int;   // Maximum cycle time of OB1 (milliseconds)
      OB1_DATE_TIME : Date_And_Time;   // Date and time OB1 started
   END_VAR
BEGIN
END_ORGANIZATION_BLOCK

// ===== PLC "JAVA"  CPU 313C-2 DP =====

ORGANIZATION_BLOCK "Main"   // OB1, LAD
TITLE = "Main Program Sweep (Cycle)"
{ S7_Optimized_Access := 'FALSE' }
VERSION : 0.1
   VAR_TEMP
      OB1_EV_CLASS : Byte;   // Bits 0-3 = 1 (Coming event), Bits 4-7 = 1 (Event class 1)
      OB1_SCAN_1 : Byte;   // 1 (Cold restart scan 1 of OB 1), 3 (Scan 2-n of OB 1)
      OB1_PRIORITY : Byte;   // Priority of OB Execution
      OB1_OB_NUMBR : Byte;   // 1 (Organization block 1, OB1)
      OB1_RESERVED_1 : Byte;   // Reserved for system
      OB1_RESERVED_2 : Byte;   // Reserved for system
      OB1_PREV_CYCLE : Int;   // Cycle time of previous OB1 scan (milliseconds)
      OB1_MIN_CYCLE : Int;   // Minimum cycle time of OB1 (milliseconds)
      OB1_MAX_CYCLE : Int;   // Maximum cycle time of OB1 (milliseconds)
      OB1_DATE_TIME : Date_And_Time;   // Date and time OB1 started
   END_VAR
BEGIN
END_ORGANIZATION_BLOCK